TYPE _00BH11_PLCTOHW_PDOS :
STRUCT
	
	outputByte_0 	 : BYTE;
	outputByte_1 	 : BYTE;

END_STRUCT
END_TYPE

(* stored: Version 1.1.0.1
   DUT _00BH11_PLCTOHW_PDOS: Id {ea5193e9-3427-46ac-bb06-ee258331e3d0} *)
